FUNCTION_BLOCK FB_Example
VAR_INPUT
    someInput               : LREAL;	// Comment
    otherInput:INT;
END_VAR
VAR_OUTPUT
END_VAR
VAR
    flag            : BOOL;
	i				: USINT;
END_VAR

FOR i := 1 TO 5 DO
			
    IF otherInput < 1.0 THEN
    	flag := (someInput < 1.0);
	END_IF


// Trailing spaces:
flag := FALSE;         

// Trailing tabs:
flag := TRUE;			

END_FOR

END_FUNCTION_BLOCK

(* stored: Version 1.1.0.1, ProductVersion 3.1.4026.17
   POU FB_Example: Id {bebb6320-5f8d-442b-bc9e-479d8a85bedf}, SpecialFunc None *)
